Yaskawa INFORM job: SHIP-R2.JBI

/JOB
//NAME SHIP-R2
//POS
///NPOS 1,0,0,0,0,0
///TOOL 1
///POSTYPE PULSE
///PULSE
C00000=2,-200297,-136925,0,-29583,0
//INST
///DATE 2023/08/08 10:17
///ATTR SC,RW
///GROUP1 RB2
NOP
MOVJ C00000 VJ=0.78
END
